(* PLC project LMM.project, Inovance company InoProShop(V1.9.1.6) InoProShop(V1.9.1.6) *)
(* stored: creationDateTime 2026-07-16T22:05:55.4194763, modificationDateTime 2026-07-16T22:05:33.9327845 *)

VAR_GLOBAL  (* GVL *)
  StartBtn AT %IX1.6 : BOOL;  (* 【面板启动】AT %IX1.6 → HMI_xStart/HMI_xEnable（上升沿 STOP→RUN） *)
  StopBtn AT %IX1.4 : BOOL;  (* 【面板停止】AT %IX1.4 → HMI_xStop *)
  ResetBtn : BOOL;  (* 【面板复位】→ HMI_xStopHold3s（错误复位脉冲）；地址现场可另绑 *)
  EStop AT %IX0.4 : BOOL;  (* 【面板急停】AT %IX0.4 正常=TRUE 按下=FALSE → 直通 HMI_xEStop *)
  StopLamp AT %QX0.6 : BOOL;  (* 【停止指示灯】AT %QX0.6 ← Dev_xStop（停止/待机） *)
  StartLamp AT %QX0.7 : BOOL;  (* 【启动/运行指示灯】AT %QX0.7 ← Dev_xRun（正在运行） *)
  JogVel : REAL;  (* 面板点动速度 → 桥接到 HMI_rJogVel* *)
  JogFwd : BOOL;  (* 面板前进 → 按 X 模式映射到 Sync/Diff/独立点动+ *)
  JogBwd : BOOL;  (* 面板后退 → 按 X 模式映射到 Sync/Diff/独立点动- *)
  JogUp : BOOL;  (* 面板上 → HMI_xJogZPos *)
  JogDown : BOOL;  (* 面板下 → HMI_xJogZNeg *)
  JogRight : BOOL;  (* 面板右 → HMI_xJogYPos *)
  JogLeft : BOOL;  (* 面板左 → HMI_xJogYNeg *)
  JogClockAdd : BOOL;  (* 顺时针 *)
  JogClockMis : BOOL;  (* 逆时针 *)
  JogACC : REAL;  (* 点动加速度 → AxisCmd_rAcc *)
  JogDEC : REAL;  (* 点动减速度 → AxisCmd_rDec *)
  HomeReq : BOOL;  (* 面板回零 → HMI_xHomeReqY/Z *)
  CaliForReq : BOOL;  (* 重力标定 *)
  ClearBruch : BOOL;  (* 毛刷清洗 *)
  yLength : REAL;  (* 龙门跨距/Y长度设定 4..6m → HMI_rWheelBase *)
  HMI_xEStop : BOOL;  (* 【急停】TRUE=未按下(正常)；FALSE=急停按下。可按可松，锁存由Logic保持 *)
  HMI_xStop : BOOL;  (* 【设备停止】短按RUN→STOP；长按3s故障复位 *)
  HMI_xStopHold3s : BOOL;  (* 【停止长按满3s脉冲】清急停锁存+轴错误复位+下使能 *)
  HMI_xEnable : BOOL;  (* 【使能/启动别名】与HMI_xStart等效；上升沿STOP→RUN *)
  Dev_xError : BOOL;  (* 【内部故障态】 *)
  Dev_xRun : BOOL;  (* 【内部运行态】 *)
  Dev_xStop : BOOL;  (* 【内部停机态】 *)
  eDevState : INT;  (* 【设备状态】0STOP 1RUN 2ERROR *)
  HMI_xDevError : BOOL;  (* 【故障灯设备级】 *)
  HMI_xDevRun : BOOL;  (* 【运行灯】 *)
  HMI_xDevStop : BOOL;  (* 【停机灯】 *)
  HMI_eOpMode : INT;  (* 【运行方式】0手动 1自动；配合Run灯 *)
  HMI_eDevState : INT;  (* 【设备状态码】0=STOP 1=RUN 2=ERROR *)
  HMI_xStart : BOOL;  (* 【设备启动】瞬时；上升沿STOP→RUN *)
  HMI_xJogYPos : BOOL;  (* 【Y点动+】TRUE移动 FALSE暂停；受限位/Z忙 *)
  HMI_xJogYNeg : BOOL;  (* 【Y点动-】TRUE移动 FALSE暂停 *)
  HMI_xJogZPos : BOOL;  (* 【Z点动+】TRUE移动 FALSE暂停 *)
  HMI_xJogZNeg : BOOL;  (* 【Z点动-】TRUE移动 FALSE暂停 *)
  HMI_xJogRPos : BOOL;  (* 【R点动+】预留；M5未就绪无效 *)
  HMI_xJogRNeg : BOOL;  (* 【R点动-】预留 *)
  HMI_rJogVelX : REAL := 0.4;  (* 【X点动速度】龙门X基速设定 *)
  AxisCmd_rSpinVel : REAL := 0.0;
  HMI_rJogVelR : REAL := 0.2;  (* 【R轴手动速度】 *)
  HMI_rSpinVel : REAL := 0.3;  (* 【X轴旋转速度】 *)
  HMI_rJogVelY : REAL := 0.4;  (* 【Y点动速度】 *)
  HMI_rJogVelZ : REAL := 0.4;  (* 【Z点动速度】 *)
  HMI_rWheelBase : REAL := 5.0;  (* 【龙门跨距=Y行程】单位m，合法范围4..6；自动Y走距用此值 *)
  xEStopLatched : BOOL;  (* 【急停锁存】按下急停置位；仅长按停止复位可清 *)
  xEnablePermit : BOOL;  (* 【使能许可】急停未触发且无锁存且无故障；≠已上使能 *)
  xFaultAggregate : BOOL;  (* 【故障汇总】任轴Fault *)
  xIlk_BlockYPlus : BOOL;  (* 【联锁禁Y+】由Y+限位派生 *)
  xIlk_BlockYNeg : BOOL;  (* 【联锁禁Y-】由Y-限位派生 *)
  xIlk_BlockZPlus : BOOL;  (* 【联锁禁Z+】由Z+限位派生 *)
  xIlk_BlockZNeg : BOOL;  (* 【联锁禁Z-】由Z-限位派生 *)
  xIlk_BlockYWhenZ : BOOL;  (* 【Z动禁Y】Z运动中禁止Y点动 *)
  xM5Ready : BOOL;  (* 【第5轴就绪】FALSE=忽略R轴 *)
  HMI_xLampEStop : BOOL;  (* 【急停灯】HMI读；锁存或按钮仍按下 *)
  HMI_xLampEnableOk : BOOL;  (* 【使能/运行灯】=设备RUN *)
  HMI_xLampFault : BOOL;  (* 【轴故障灯】 *)
  eOpMode : INT;  (* 【运行模式】0=手动Manual（本期固定） *)
  iAlarmID : INT;  (* 【内部报警号】Logic判定后拷贝到HMI_iAlarmShow *)
  HMI_iAlarmShow : INT;  (* 【报警号】0无；1001急停；1002故障；1003限位；1004无许可；1099R未就绪 *)
  I_xLimYPos : BOOL;  (* 【Y正限位】物理输入，地址%I* TBD *)
  I_xLimYNeg : BOOL;  (* 【Y负限位】物理输入 *)
  I_xHomeY : BOOL;  (* 【Y原点】物理输入 *)
  I_xLimZPos : BOOL;  (* 【Z正限位】物理输入 *)
  I_xLimZNeg : BOOL;  (* 【Z负限位】物理输入 *)
  I_xHomeZ : BOOL;  (* 【Z原点】物理输入 *)
  I_xLimRPos : BOOL;  (* 【R正限位】预留 *)
  I_xLimRNeg : BOOL;  (* 【R负限位】预留 *)
  I_xHomeR : BOOL;  (* 【R原点】预留 *)
  AxisCmd_xPower : BOOL;  (* 【轴使能命令】仅设备RUN时TRUE *)
  AxisCmd_xJogYPos : BOOL;  (* 【Y点动+命令】含限位/Z忙门控 *)
  AxisCmd_xJogYNeg : BOOL;  (* 【Y点动-命令】 *)
  AxisCmd_xJogZPos : BOOL;  (* 【Z点动+命令】 *)
  AxisCmd_xJogZNeg : BOOL;  (* 【Z点动-命令】 *)
  AxisCmd_xJogRPos : BOOL;  (* 【R点动+命令】预留 *)
  AxisCmd_xJogRNeg : BOOL;  (* 【R点动-命令】预留 *)
  AxisCmd_xStopAll : BOOL;  (* 【全停】急停/停止/故障时TRUE *)
  AxisCmd_xResetFault : BOOL;  (* 【错误复位脉冲】一拍TRUE→各轴MC_Reset *)
  AxisCmd_rWheelBase : REAL;  (* 【跨距L命令】限幅4..6m *)
  AxisCmd_rJogVelX : REAL;  (* 【X点动速度命令】 *)
  AxisCmd_rJogVelY : REAL;  (* 【Y点动速度命令】 *)
  AxisCmd_rJogVelZ : REAL;  (* 【Z点动速度命令】 *)
  AxisCmd_rJogVelR : REAL;  (* 【R点动速度命令】预留 *)
  AxisCmd_rAcc : REAL;  (* 【加速度】 *)
  AxisCmd_rDec : REAL;  (* 【减速度】 *)
  AxisFb_rVelCmdM1 : REAL;  (* 【M1速度指令反馈】供HMI显示 *)
  AxisFb_rVelCmdM2 : REAL;  (* 【M2速度指令反馈】 *)
  AxisFb_rPosM1 : REAL;  (* 【M1实际位置】 *)
  AxisFb_rPosM2 : REAL;  (* 【M2实际位置】 *)
  AxisFb_rPosY : REAL;  (* 【Y实际位置】 *)
  AxisFb_rPosZ : REAL;  (* 【Z实际位置】 *)
  AxisFb_rPosR : REAL;  (* 【R实际位置】预留 *)
  AxisFb_xStandstill1 : BOOL;  (* 【M1静止】 *)
  AxisFb_xStandstill2 : BOOL;  (* 【M2静止】 *)
  AxisFb_xStandstillY : BOOL;  (* 【Y静止】 *)
  AxisFb_xStandstillZ : BOOL;  (* 【Z静止】 *)
  AxisFb_xStandstillR : BOOL;  (* 【R静止】预留 *)
  AxisFb_xMovingM1 : BOOL;  (* 【M1运动中】 *)
  AxisFb_xMovingM2 : BOOL;  (* 【M2运动中】 *)
  AxisFb_xMovingY : BOOL;  (* 【Y运动中】 *)
  AxisFb_xMovingZ : BOOL;  (* 【Z运动中】 *)
  AxisFb_xMovingR : BOOL;  (* 【R运动中】预留 *)
  AxisFb_xPoweredM1 : BOOL;  (* 【M1已使能】驱动功率级就绪，HMI灯 *)
  AxisFb_xPoweredM2 : BOOL;  (* 【M2已使能】 *)
  AxisFb_xPoweredY : BOOL;  (* 【Y已使能】 *)
  AxisFb_xPoweredZ : BOOL;  (* 【Z已使能】 *)
  AxisFb_xPoweredR : BOOL;  (* 【R已使能】预留 *)
  AxisFb_xHomedY : BOOL;  (* 【Y已回零】 *)
  AxisFb_xHomedZ : BOOL;  (* 【Z已回零】 *)
  AxisFb_xHomedR : BOOL;  (* 【R已回零】预留 *)
  AxisFb_xFaultM1 : BOOL;  (* 【M1故障】 *)
  AxisFb_xFaultM2 : BOOL;  (* 【M2故障】 *)
  AxisFb_xFaultY : BOOL;  (* 【Y故障】 *)
  AxisFb_xFaultZ : BOOL;  (* 【Z故障】 *)
  AxisFb_xFaultR : BOOL;  (* 【R故障】预留 *)
  AxisFb_xReady : BOOL;  (* 【轴就绪】四轴无故障、可参与运动 *)
  HMI_xAutoMode : BOOL;  (* 【自动模式】TRUE自动 FALSE手动 *)
  HMI_xJogXPos : BOOL;  (* 【X+】同步直行 *)
  HMI_xJogXNeg : BOOL;  (* 【X-】 *)
  HMI_xSpinLeft : BOOL;  (* 【左旋转】 *)
  HMI_xSpinRight : BOOL;  (* 【右旋转】 *)
  HMI_xAutoStart : BOOL;  (* 【自动启动】 *)
  HMI_xAutoAbort : BOOL;  (* 【自动中止】 *)
  HMI_rAutoDistX : REAL;  (* 【自动X距离】 *)
  HMI_rAutoVelX : REAL;  (* 【自动X速度】 *)
  HMI_rAutoVelY : REAL;  (* 【自动Y速度】 *)
  HMI_rAutoVelZ : REAL;  (* 【自动Z速度】 *)
  HMI_rForceSet : REAL;  (* 【力设定N】 *)
  HMI_xForceSimEnable : BOOL;  (* 【力模拟使能】 *)
  HMI_rForceSim : REAL;  (* 【力模拟值N】 *)
  HMI_iAutoStepShow : INT;  (* 【自动步号】 *)
  HMI_xAutoBusy : BOOL;  (* 【自动忙】 *)
  HMI_xAutoDone : BOOL;  (* 【自动完成】 *)
  HMI_rForceShow : REAL;  (* 【力实际N】 *)
  Tcp_xConnected : BOOL;  (* 【TCP】已连接 *)
  Tcp_xTimeout : BOOL;  (* 【TCP】通讯超时 *)
  Tcp_xOnline : BOOL;  (* 【TCP】Connected且未超时 *)
  Tcp_xEStop : BOOL := TRUE;  (* 【TCP急停影子】默认TRUE；与面板AND合成 *)
  Tcp_xStop : BOOL;
  Tcp_xStopHold3s : BOOL;
  Tcp_xStart : BOOL;
  Tcp_xEnable : BOOL;
  Tcp_xAutoMode : BOOL;
  Tcp_xJogXPos : BOOL;
  Tcp_xJogXNeg : BOOL;
  Tcp_xSpinLeft : BOOL;
  Tcp_xSpinRight : BOOL;
  Tcp_xJogYPos : BOOL;
  Tcp_xJogYNeg : BOOL;
  Tcp_xJogZPos : BOOL;
  Tcp_xJogZNeg : BOOL;
  Tcp_xJogRPos : BOOL;
  Tcp_xJogRNeg : BOOL;
  Tcp_rJogVelX : REAL := 0.4;
  Tcp_rSpinVel : REAL := 0.3;
  Tcp_rJogVelY : REAL := 0.3;
  Tcp_rJogVelZ : REAL := 0.2;
  Tcp_rJogVelR : REAL := 0.2;
  Tcp_xAutoStart : BOOL;
  Tcp_xAutoAbort : BOOL;
  Tcp_rAutoDistX : REAL := 1.0;
  Tcp_rAutoVelX : REAL := 0.4;
  Tcp_rAutoVelY : REAL := 0.3;
  Tcp_rAutoVelZ : REAL := 0.15;
  Tcp_rWheelBase : REAL := 5.0;
  Tcp_rForceSet : REAL := 100.0;
  Tcp_xForceSimEnable : BOOL := TRUE;
  Tcp_rForceSim : REAL;
  Tcp_uiPort : UINT := 9100;  (* 【TCP监听端口】默认9100 *)
  iAutoStep : INT;  (* 【自动步】0Idle..5Done *)
  rForceAct : REAL;  (* 【实际力N】 *)
  rForceKp : REAL;  (* 【恒力Kp】 *)
  AxisCmd_xJogXPos : BOOL;  (* 【Axis X+】 *)
  AxisCmd_xJogXNeg : BOOL;  (* 【Axis X-】 *)
  AxisCmd_xSpinLeft : BOOL;  (* 【Axis 左旋】 *)
  AxisCmd_xSpinRight : BOOL;  (* 【Axis 右旋】 *)
  AxisCmd_xMoveRelX : BOOL;  (* 【Axis X相对】 *)
  AxisCmd_rMoveDistX : REAL;  (* 【X相对距离】 *)
  AxisCmd_rMoveVelX : REAL;  (* 【X相对速度】 *)
  AxisCmd_xMoveRelY : BOOL;  (* 【Axis Y相对】 *)
  AxisCmd_rMoveDistY : REAL;  (* 【Y相对距离】 *)
  AxisCmd_rMoveVelY : REAL;  (* 【Y相对速度】 *)
  AxisCmd_rZVelCmd : REAL;  (* 【Z速度指令】 *)
  AxisCmd_xUseZVelCmd : BOOL;  (* 【使用Z速度指令】 *)
  AxisCmd_xHoldR : BOOL;  (* 【R保持】 *)
  AxisCmd_rRHoldPos : REAL;  (* 【R保持角】 *)
  AxisFb_xMoveDoneX : BOOL;  (* 【X相对到位】 *)
  AxisFb_xMoveDoneY : BOOL;  (* 【Y相对到位】 *)
END_VAR

PROGRAM PRG_Axis_Control
  VAR
    fbM1 : FB_Servo;
    fbM2 : FB_Servo;
    fbY : FB_Servo;
    fbZ : FB_Servo;
    fbXDiff : FB_XDiff;
    xPair : BOOL;
    eModeX : INT;
    xDiffPos : BOOL;
    xDiffNeg : BOOL;
    rXVel : REAL;
  END_VAR

            (*==============================================================================
 * PRG_Axis_Control — 运动独立任务（AxisTask）
 * 仅通过 GVL_AxisCmd 输入 / GVL_AxisFb 输出；禁止被外部 CALL
 * 轴绑定：Axis=M1, Axis_1=M2, Axis_2=Y, Axis_3=Z
 *============================================================================*)

(* X：同步直行 / 左右旋；VelX 与 SpinVel 分开 *)
eModeX := 0;
xDiffPos := FALSE; xDiffNeg := FALSE;
IF AxisCmd_xSpinLeft XOR AxisCmd_xSpinRight THEN
	eModeX := 2;
	xDiffPos := AxisCmd_xSpinLeft;
	xDiffNeg := AxisCmd_xSpinRight;
	rXVel := AxisCmd_rSpinVel;
ELSIF AxisCmd_xJogXPos XOR AxisCmd_xJogXNeg THEN
	eModeX := 1;
	rXVel := AxisCmd_rJogVelX;
ELSE
	rXVel := 0.0;
END_IF;

fbXDiff(
	eMode := eModeX,
	eDiffFunc := 1,
	xJogSyncPos := AxisCmd_xJogXPos,
	xJogSyncNeg := AxisCmd_xJogXNeg,
	xJogDiffPos := xDiffPos,
	xJogDiffNeg := xDiffNeg,
	xStop := AxisCmd_xStopAll,
	xEnable := AxisCmd_xPower,
	rJogVel := rXVel,
	rDiffDelta := 0.0,
	rTurnOmega := 0.0,
	rWheelBase := AxisCmd_rWheelBase
);
xPair := fbXDiff.xUsePairVel;

IF xPair THEN
	(* 成对模式：用 FB_XDiff 输出的有符号速度 *)
	fbM1(
		Axis := _MC_Axis[1],
		xEnable := AxisCmd_xPower,
		xJogPos := FALSE, xJogNeg := FALSE,
		xStop := AxisCmd_xStopAll,
		xResetFault := AxisCmd_xResetFault,
		xHome := FALSE,
		xUseVelCmd := TRUE,
		rVelCmd := fbXDiff.rVelCmdM1,
		rJogVel := rXVel,
		rAcc := AxisCmd_rAcc,
		rDec := AxisCmd_rDec
	);
	fbM2(
		Axis := _MC_Axis[2],
		xEnable := AxisCmd_xPower,
		xJogPos := FALSE, xJogNeg := FALSE,
		xStop := AxisCmd_xStopAll,
		xResetFault := AxisCmd_xResetFault,
		xHome := FALSE,
		xUseVelCmd := TRUE,
		rVelCmd := fbXDiff.rVelCmdM2,
		rJogVel := rXVel,
		rAcc := AxisCmd_rAcc,
		rDec := AxisCmd_rDec
	);
	AxisFb_rVelCmdM1 := fbXDiff.rVelCmdM1;
	AxisFb_rVelCmdM2 := fbXDiff.rVelCmdM2;
ELSE
	(* 无 X 命令：两侧保持上电待机 *)
	fbM1(
		Axis := _MC_Axis[1],
		xEnable := AxisCmd_xPower,
		xJogPos := FALSE, xJogNeg := FALSE,
		xStop := AxisCmd_xStopAll,
		xResetFault := AxisCmd_xResetFault,
		xHome := FALSE,
		xUseVelCmd := FALSE,
		rVelCmd := 0.0,
		rJogVel := AxisCmd_rJogVelX,
		rAcc := AxisCmd_rAcc,
		rDec := AxisCmd_rDec
	);
	fbM2(
		Axis := _MC_Axis[2],
		xEnable := AxisCmd_xPower,
		xJogPos := FALSE, xJogNeg := FALSE,
		xStop := AxisCmd_xStopAll,
		xResetFault := AxisCmd_xResetFault,
		xHome := FALSE,
		xUseVelCmd := FALSE,
		rVelCmd := 0.0,
		rJogVel := AxisCmd_rJogVelX,
		rAcc := AxisCmd_rAcc,
		rDec := AxisCmd_rDec
	);
	AxisFb_rVelCmdM1 := 0.0;
	AxisFb_rVelCmdM2 := 0.0;
END_IF;

(* Y / Z *)
fbY(
	Axis := _MC_Axis[3],
	xEnable := AxisCmd_xPower,
	xJogPos := AxisCmd_xJogYPos,
	xJogNeg := AxisCmd_xJogYNeg,
	xStop := AxisCmd_xStopAll,
	xResetFault := AxisCmd_xResetFault,
	xHome := FALSE,
	xUseVelCmd := FALSE,
	rVelCmd := 0.0,
	rJogVel := AxisCmd_rJogVelY,
	rAcc := AxisCmd_rAcc,
	rDec := AxisCmd_rDec
);
fbZ(
	Axis := _MC_Axis[4],
	xEnable := AxisCmd_xPower,
	xJogPos := AxisCmd_xJogZPos,
	xJogNeg := AxisCmd_xJogZNeg,
	xStop := AxisCmd_xStopAll,
	xResetFault := AxisCmd_xResetFault,
	xHome := FALSE,
	xUseVelCmd := FALSE,
	rVelCmd := 0.0,
	rJogVel := AxisCmd_rJogVelZ,
	rAcc := AxisCmd_rAcc,
	rDec := AxisCmd_rDec
);

(* ---------- 写反馈区（仅本任务可写） ---------- *)
AxisFb_rPosM1 := fbM1.rActPos;
AxisFb_rPosM2 := fbM2.rActPos;
AxisFb_rPosY := fbY.rActPos;
AxisFb_rPosZ := fbZ.rActPos;
AxisFb_xMovingM1 := fbM1.xMoving;
AxisFb_xMovingM2 := fbM2.xMoving;
AxisFb_xMovingY := fbY.xMoving;
AxisFb_xMovingZ := fbZ.xMoving;
AxisFb_xPoweredM1 := fbM1.xPowered;
AxisFb_xPoweredM2 := fbM2.xPowered;
AxisFb_xPoweredY := fbY.xPowered;
AxisFb_xPoweredZ := fbZ.xPowered;
AxisFb_xFaultM1 := fbM1.xFault;
AxisFb_xFaultM2 := fbM2.xFault;
AxisFb_xFaultY := fbY.xFault;
AxisFb_xFaultZ := fbZ.xFault;
AxisFb_xHomedY := fbY.xHomed;
AxisFb_xHomedZ := fbZ.xHomed;
AxisFb_xStandstill1 := fbM1.xStandstill;
AxisFb_xStandstill2 := fbM2.xStandstill;
AxisFb_xStandstillY := fbY.xStandstill;
AxisFb_xStandstillZ := fbZ.xStandstill;
AxisFb_xReady := NOT (fbM1.xFault OR fbM2.xFault OR fbY.xFault OR fbZ.xFault);

          
END_PROGRAM

FUNCTION_BLOCK FB_XDiff
  VAR_INPUT
    eMode : INT;
    eDiffFunc : INT;
    xJogSyncPos : BOOL;
    xJogSyncNeg : BOOL;
    xJogDiffPos : BOOL;
    xJogDiffNeg : BOOL;
    xStop : BOOL;
    xEnable : BOOL;
    rJogVel : REAL;
    rDiffDelta : REAL;
    rTurnOmega : REAL;
    rWheelBase : REAL;
  END_VAR
  VAR_OUTPUT
    rVelCmdM1 : REAL;
    rVelCmdM2 : REAL;
    xActive : BOOL;
    xUsePairVel : BOOL;
    xWheelBaseOk : BOOL;
  END_VAR

            (*==============================================================================
 * FB_XDiff — 龙门 X 双驱速度合成（仅 Axis 任务内使用）
 * eMode: 0=独立  1=同步同速平移  2=差速（子功能见 eDiffFunc）
 * eDiffFunc: 0=纠偏  1=原地旋转(一正一反)  2=差速拐弯
 * 跨距 rWheelBase: 4..6 m；X 运动方向与 Y 垂直
 *============================================================================*)

(* 输出清零 *)
rVelCmdM1 := 0.0;
rVelCmdM2 := 0.0;
xUsePairVel := FALSE;
xActive := FALSE;
(* 跨距合法性 *)
xWheelBaseOk := (rWheelBase >= 4.0) AND (rWheelBase <= 6.0);

(* 未使能 / 停止 / 独立模式：不合成成对速度 *)
IF NOT xEnable OR xStop OR eMode = 0 THEN
	RETURN;
END_IF;

(* ---------- Sync：两侧同速，龙门沿 X 平移 ---------- *)
IF eMode = 1 THEN
	IF xJogSyncPos XOR xJogSyncNeg THEN
		xUsePairVel := TRUE;
		xActive := TRUE;
		IF xJogSyncPos THEN
			rVelCmdM1 := rJogVel;
		ELSE
			rVelCmdM1 := -rJogVel;
		END_IF;
		rVelCmdM2 := rVelCmdM1; (* 同速 *)
	END_IF;
	RETURN;
END_IF;

(* ---------- Diff：需有方向键 ---------- *)
IF NOT (xJogDiffPos XOR xJogDiffNeg) THEN
	RETURN;
END_IF;

(* 原地旋转 / 差速拐弯依赖合法跨距 *)
IF (eDiffFunc = 1 OR eDiffFunc = 2) AND NOT xWheelBaseOk THEN
	RETURN;
END_IF;

xUsePairVel := TRUE;
xActive := TRUE;

CASE eDiffFunc OF
	0: (* 纠偏：同向 V±Δ，扶正龙门 *)
		IF xJogDiffPos THEN
			rVelCmdM1 := rJogVel + rDiffDelta;
			rVelCmdM2 := rJogVel - rDiffDelta;
		ELSE
			rVelCmdM1 := -(rJogVel + rDiffDelta);
			rVelCmdM2 := -(rJogVel - rDiffDelta);
		END_IF;

	1: (* 原地旋转：M1/M2 一正一反，转角度 *)
		IF ABS(rTurnOmega) > 1.0E-6 THEN
			rVelCmdM1 := rTurnOmega * rWheelBase * 0.5;
		ELSE
			rVelCmdM1 := rJogVel;
		END_IF;
		rVelCmdM2 := -rVelCmdM1;
		IF xJogDiffNeg THEN
			rVelCmdM1 := -rVelCmdM1;
			rVelCmdM2 := -rVelCmdM2;
		END_IF;

	2: (* 差速拐弯：两侧同向为主，速度差，可边走边弯 *)
		IF ABS(rTurnOmega) > 1.0E-6 THEN
			rVelCmdM1 := rJogVel + rTurnOmega * rWheelBase * 0.5;
			rVelCmdM2 := rJogVel - rTurnOmega * rWheelBase * 0.5;
		ELSE
			rVelCmdM1 := rJogVel + rDiffDelta;
			rVelCmdM2 := rJogVel - rDiffDelta;
		END_IF;
		IF xJogDiffNeg THEN
			rVelCmdM1 := -rVelCmdM1;
			rVelCmdM2 := -rVelCmdM2;
		END_IF;

ELSE
	xUsePairVel := FALSE;
	xActive := FALSE;
END_CASE;

          
END_FUNCTION_BLOCK

PROGRAM PLC_PRG

            (*==============================================================================
 * PLC_PRG — 主任务入口（MainTask）
 * 只调用逻辑程序；禁止在此 CALL PRG_Axis_Control（轴控在独立 AxisTask）
 *============================================================================*)
PRG_TcpHmi();
PRG_Logic();

          
END_PROGRAM

PROGRAM PRG_Logic
  VAR
    tonHold : TON;
    tonResetHold : TON;
    xResetPulse : BOOL;
    xResetPrev : BOOL;
    xStartEdge : BOOL;
    xStartPrev : BOOL;
    xStopEdge : BOOL;
    xStopPrev : BOOL;
    xPostResetHold : BOOL;
    xAutoStartPrev : BOOL;
    xAutoStartEdge : BOOL;
    rRHold : REAL;
    xMoveXSent : BOOL;
    xMoveYSent : BOOL;
    xBridgeInited : BOOL;
  END_VAR

            (*==============================================================================
 * PRG_Logic — 设备态 / 手动裁定 / 自动步序 / 恒力
 * 禁止 CALL Axis / FB_Servo / FB_XDiff
 *============================================================================*)

(* —— 面板 ∨ TCP 影子 → HMI（见 docs/plc/TCP_HMI.md）—— *)
Tcp_xOnline := Tcp_xConnected AND NOT Tcp_xTimeout;
HMI_xEStop := EStop AND Tcp_xEStop;
HMI_xStop := StopBtn OR Tcp_xStop;
HMI_xStart := StartBtn OR Tcp_xStart;
HMI_xEnable := StartBtn OR Tcp_xEnable OR Tcp_xStart;
HMI_xStopHold3s := ResetBtn OR Tcp_xStopHold3s;
IF Tcp_xOnline THEN
	HMI_xAutoMode := Tcp_xAutoMode;
	HMI_xForceSimEnable := Tcp_xForceSimEnable;
END_IF;
HMI_xJogXPos := JogFwd OR Tcp_xJogXPos;
HMI_xJogXNeg := JogBwd OR Tcp_xJogXNeg;
HMI_xSpinLeft := Tcp_xSpinLeft;
HMI_xSpinRight := Tcp_xSpinRight;
HMI_xJogYPos := JogRight OR Tcp_xJogYPos;
HMI_xJogYNeg := JogLeft OR Tcp_xJogYNeg;
HMI_xJogZPos := JogUp OR Tcp_xJogZPos;
HMI_xJogZNeg := JogDown OR Tcp_xJogZNeg;
HMI_xJogRPos := Tcp_xJogRPos;
HMI_xJogRNeg := Tcp_xJogRNeg;
HMI_xAutoStart := Tcp_xAutoStart;
HMI_xAutoAbort := Tcp_xAutoAbort;
IF Tcp_xOnline THEN
	HMI_rJogVelX := Tcp_rJogVelX;
	HMI_rSpinVel := Tcp_rSpinVel;
	HMI_rJogVelY := Tcp_rJogVelY;
	HMI_rJogVelZ := Tcp_rJogVelZ;
	HMI_rJogVelR := Tcp_rJogVelR;
	HMI_rAutoDistX := Tcp_rAutoDistX;
	HMI_rAutoVelX := Tcp_rAutoVelX;
	HMI_rAutoVelY := Tcp_rAutoVelY;
	HMI_rAutoVelZ := Tcp_rAutoVelZ;
	HMI_rWheelBase := Tcp_rWheelBase;
	HMI_rForceSet := Tcp_rForceSet;
	HMI_rForceSim := Tcp_rForceSim;
ELSE
	HMI_rJogVelX := JogVel;
	HMI_rJogVelY := JogVel;
	HMI_rJogVelZ := JogVel;
END_IF;

(* —— 急停 / 复位 —— *)
IF NOT HMI_xEStop THEN xEStopLatched := TRUE; END_IF;
tonHold(IN := HMI_xStop AND HMI_xEStop, PT := T#3S);
xResetPulse := (HMI_xStopHold3s OR tonHold.Q) AND NOT xResetPrev;
xResetPrev := HMI_xStopHold3s OR tonHold.Q;
IF xResetPulse THEN
	xEStopLatched := FALSE;
	AxisCmd_xResetFault := TRUE;
	eDevState := 0;
	xPostResetHold := TRUE;
	iAutoStep := 0;
ELSE
	AxisCmd_xResetFault := FALSE;
END_IF;

xFaultAggregate := AxisFb_xFaultM1 OR AxisFb_xFaultM2 OR AxisFb_xFaultY OR AxisFb_xFaultZ
	OR (xM5Ready AND AxisFb_xFaultR);
xEnablePermit := HMI_xEStop AND NOT xEStopLatched AND NOT xFaultAggregate;
IF HMI_xAutoMode THEN eOpMode := 1; ELSE eOpMode := 0; END_IF;
HMI_eOpMode := eOpMode;

tonResetHold(IN := xPostResetHold, PT := T#2S);
IF NOT xFaultAggregate AND HMI_xEStop AND NOT xEStopLatched THEN
	xPostResetHold := FALSE;
ELSIF tonResetHold.Q OR NOT HMI_xEStop OR xEStopLatched THEN
	xPostResetHold := FALSE;
END_IF;

xStartEdge := (HMI_xStart OR HMI_xEnable) AND NOT xStartPrev;
xStartPrev := HMI_xStart OR HMI_xEnable;
xStopEdge := HMI_xStop AND NOT xStopPrev;
xStopPrev := HMI_xStop;

IF xResetPulse THEN
	eDevState := 0;
ELSIF NOT HMI_xEStop OR xEStopLatched THEN
	eDevState := 2;
ELSIF xFaultAggregate AND NOT xPostResetHold THEN
	eDevState := 2;
ELSIF eDevState = 2 THEN
	;
ELSIF xStopEdge AND NOT tonHold.Q THEN
	eDevState := 0;
	iAutoStep := 0;
ELSIF xStartEdge AND eDevState = 0 AND xEnablePermit THEN
	eDevState := 1;
ELSIF xStartEdge AND eDevState = 0 AND NOT xEnablePermit THEN
	iAlarmID := 1004;
END_IF;

Dev_xStop := (eDevState = 0);
Dev_xRun := (eDevState = 1);
Dev_xError := (eDevState = 2);
HMI_eDevState := eDevState;
HMI_xDevStop := Dev_xStop;
HMI_xDevRun := Dev_xRun;
HMI_xDevError := Dev_xError;

IF HMI_xForceSimEnable THEN
	rForceAct := HMI_rForceSim;
END_IF;
HMI_rForceShow := rForceAct;
IF rForceKp < 1.0E-6 THEN rForceKp := 1.0; END_IF;

xIlk_BlockYPlus := I_xLimYPos; xIlk_BlockYNeg := I_xLimYNeg;
xIlk_BlockZPlus := I_xLimZPos; xIlk_BlockZNeg := I_xLimZNeg;
xIlk_BlockYWhenZ := FALSE;

AxisCmd_xStopAll := (eDevState <> 1) OR HMI_xStop OR HMI_xAutoAbort;
AxisCmd_xPower := (eDevState = 1);
AxisCmd_rJogVelX := HMI_rJogVelX;
AxisCmd_rSpinVel := HMI_rSpinVel;
AxisCmd_rJogVelY := HMI_rJogVelY;
AxisCmd_rJogVelZ := HMI_rJogVelZ;
AxisCmd_rJogVelR := HMI_rJogVelR;
AxisCmd_rWheelBase := LIMIT(4.0, HMI_rWheelBase, 6.0);
AxisCmd_rAcc := JogACC;
AxisCmd_rDec := JogDEC;
IF AxisCmd_rAcc < 1.0 THEN AxisCmd_rAcc := 100.0; END_IF;
IF AxisCmd_rDec < 1.0 THEN AxisCmd_rDec := 100.0; END_IF;

AxisCmd_xJogXPos := FALSE; AxisCmd_xJogXNeg := FALSE;
AxisCmd_xSpinLeft := FALSE; AxisCmd_xSpinRight := FALSE;
AxisCmd_xJogYPos := FALSE; AxisCmd_xJogYNeg := FALSE;
AxisCmd_xJogZPos := FALSE; AxisCmd_xJogZNeg := FALSE;
AxisCmd_xJogRPos := FALSE; AxisCmd_xJogRNeg := FALSE;
AxisCmd_xUseZVelCmd := FALSE; AxisCmd_rZVelCmd := 0.0;
AxisCmd_xMoveRelX := FALSE; AxisCmd_xMoveRelY := FALSE;
AxisCmd_xHoldR := FALSE;

xAutoStartEdge := HMI_xAutoStart AND NOT xAutoStartPrev;
xAutoStartPrev := HMI_xAutoStart;

IF Dev_xError OR HMI_xAutoAbort OR (eDevState <> 1) THEN
	iAutoStep := 0;
	HMI_xAutoBusy := FALSE;
END_IF;

(* ===== 手动：仅 RUN + 手动模式 ===== *)
IF Dev_xRun AND (eOpMode = 0) AND NOT HMI_xStop THEN
	IF HMI_xSpinLeft XOR HMI_xSpinRight THEN
		AxisCmd_xSpinLeft := HMI_xSpinLeft;
		AxisCmd_xSpinRight := HMI_xSpinRight;
	ELSIF HMI_xJogXPos XOR HMI_xJogXNeg THEN
		AxisCmd_xJogXPos := HMI_xJogXPos;
		AxisCmd_xJogXNeg := HMI_xJogXNeg;
	END_IF;
	AxisCmd_xJogYPos := HMI_xJogYPos AND NOT xIlk_BlockYPlus;
	AxisCmd_xJogYNeg := HMI_xJogYNeg AND NOT xIlk_BlockYNeg;
	AxisCmd_xJogZPos := HMI_xJogZPos AND NOT xIlk_BlockZPlus;
	AxisCmd_xJogZNeg := HMI_xJogZNeg AND NOT xIlk_BlockZNeg;
	IF xM5Ready THEN
		AxisCmd_xJogRPos := HMI_xJogRPos;
		AxisCmd_xJogRNeg := HMI_xJogRNeg;
	END_IF;
END_IF;

(* ===== 自动 ===== *)
IF Dev_xRun AND (eOpMode = 1) AND NOT HMI_xStop THEN
	IF iAutoStep = 0 AND xAutoStartEdge THEN
		iAutoStep := 1;
		rRHold := AxisFb_rPosR;
		xMoveXSent := FALSE; xMoveYSent := FALSE;
		HMI_xAutoDone := FALSE;
		HMI_xAutoBusy := TRUE;
	END_IF;

	CASE iAutoStep OF
		1: (* MoveX *)
			AxisCmd_xHoldR := TRUE;
			AxisCmd_rRHoldPos := rRHold;
			AxisCmd_rMoveDistX := HMI_rAutoDistX;
			AxisCmd_rMoveVelX := HMI_rAutoVelX;
			AxisCmd_xMoveRelX := TRUE;
			IF AxisFb_xMoveDoneX THEN
				AxisCmd_xMoveRelX := FALSE;
				iAutoStep := 2;
			END_IF;
		2: (* PressZ *)
			AxisCmd_xHoldR := TRUE;
			AxisCmd_rRHoldPos := rRHold;
			AxisCmd_xUseZVelCmd := TRUE;
			IF rForceAct >= HMI_rForceSet THEN
				AxisCmd_rZVelCmd := 0.0;
				iAutoStep := 3;
				xMoveYSent := FALSE;
			ELSE
				AxisCmd_rZVelCmd := -ABS(HMI_rAutoVelZ);
			END_IF;
		3: (* MoveY + 恒力 *)
			AxisCmd_xHoldR := TRUE;
			AxisCmd_rRHoldPos := rRHold;
			AxisCmd_rMoveDistY := AxisCmd_rWheelBase;
			AxisCmd_rMoveVelY := HMI_rAutoVelY;
			AxisCmd_xMoveRelY := TRUE;
			AxisCmd_xUseZVelCmd := TRUE;
			AxisCmd_rZVelCmd := LIMIT(-ABS(HMI_rAutoVelZ),
				rForceKp * (HMI_rForceSet - rForceAct), ABS(HMI_rAutoVelZ));
			IF AxisFb_xMoveDoneY THEN
				AxisCmd_xMoveRelY := FALSE;
				AxisCmd_rZVelCmd := 0.0;
				iAutoStep := 4;
			END_IF;
		4: (* RWobble 占位 *)
			iAutoStep := 5;
		5: (* Done *)
			HMI_xAutoBusy := FALSE;
			HMI_xAutoDone := TRUE;
			iAutoStep := 0;
	END_CASE;
END_IF;

IF Dev_xError THEN
	IF xEStopLatched OR NOT HMI_xEStop THEN
		iAlarmID := 1001;
	ELSE
		iAlarmID := 1002;
	END_IF;
ELSIF iAlarmID <> 1004 THEN
	iAlarmID := 0;
END_IF;

HMI_iAutoStepShow := iAutoStep;
HMI_xLampEStop := xEStopLatched OR NOT HMI_xEStop;
HMI_xLampEnableOk := Dev_xRun;
HMI_xLampFault := xFaultAggregate;
HMI_iAlarmShow := iAlarmID;

StopLamp := Dev_xStop;
StartLamp := Dev_xRun;

          
END_PROGRAM

FUNCTION_BLOCK FB_Servo
  VAR_INPUT
    xEnable : BOOL;
    xJogPos : BOOL;
    xJogNeg : BOOL;
    xStop : BOOL;
    xResetFault : BOOL;
    xHome : BOOL;
    xUseVelCmd : BOOL;
    rVelCmd : REAL;
    rJogVel : REAL;
    rAcc : REAL;
    rDec : REAL;
  END_VAR
  VAR_OUTPUT
    xPowered : BOOL;
    xMoving : BOOL;
    xStandstill : BOOL;
    xHomed : BOOL;
    xFault : BOOL;
    rActPos : LREAL;
  END_VAR
  VAR_IN_OUT
    Axis : AXIS_REF_SM3;
  END_VAR
  VAR
    fbPower : MC_Power;
    fbJog : MC_MoveVelocity;
    fbStop : MC_Stop;
    fbHome : MC_Home;
    fbReset : MC_Reset;
    fbReadStatus : MC_ReadStatus;
    fbReadPos : MC_ReadActualPosition;
    xEnInternal : BOOL;
  END_VAR

            (* 读轴状态 / 实际位置 *)
fbReadStatus(Axis := Axis, Enable := TRUE);
fbReadPos(Axis := Axis, Enable := TRUE);

rActPos := fbReadPos.Position;
xStandstill := fbReadStatus.StandStill;
xMoving := fbReadStatus.DiscreteMotion OR fbReadStatus.ContinuousMotion;

(* 故障汇总：Errorstop + 各 FB.Error（不用 Axis.bError / Operational） *)
xFault := fbReadStatus.Errorstop
	OR fbReadStatus.Error
	OR fbPower.Error
	OR fbJog.Error
	OR fbStop.Error
	OR fbReset.Error;

(* 错误复位脉冲（来自停止钮长按 3s → AxisCmd_xResetFault） *)
fbReset(Axis := Axis, Execute := xResetFault);

(* 内部使能：请求使能且未停且非 Errorstop *)
xEnInternal := xEnable AND NOT xStop AND NOT fbReadStatus.Errorstop;

(* 功率级：Enable 恒 TRUE 以刷新；实际开/关看 bRegulatorOn/bDriveStart *)
fbPower(
	Axis := Axis,
	Enable := TRUE,
	bRegulatorOn := xEnInternal,
	bDriveStart := xEnInternal
);
(* Status=TRUE 表示轴可运动 *)
xPowered := fbPower.Status;

(* ---------- 运动仲裁 ---------- *)
IF xStop OR NOT xEnable OR fbReadStatus.Errorstop THEN
	(* 停止 / 禁使能 / 故障：停速度指令并减速停 *)
	fbJog(Axis := Axis, Execute := FALSE);
	fbHome(Axis := Axis, Execute := FALSE);
	fbStop(Axis := Axis, Execute := TRUE, Deceleration := rDec);

ELSIF xHome THEN
	(* 回零 *)
	fbStop(Axis := Axis, Execute := FALSE);
	fbJog(Axis := Axis, Execute := FALSE);
	fbHome(Axis := Axis, Execute := TRUE);

ELSIF xUseVelCmd THEN
	(* 成对速度模式：使用有符号 rVelCmd（来自 FB_XDiff） *)
	fbStop(Axis := Axis, Execute := FALSE);
	fbHome(Axis := Axis, Execute := FALSE);
	IF ABS(rVelCmd) > 1.0E-6 AND xPowered THEN
		fbJog(Axis := Axis, Execute := TRUE, Velocity := rVelCmd, Acceleration := rAcc, Deceleration := rDec);
	ELSE
		fbJog(Axis := Axis, Execute := FALSE);
	END_IF;

ELSIF xJogPos XOR xJogNeg THEN
	(* 独立 JOG *)
	fbStop(Axis := Axis, Execute := FALSE);
	fbHome(Axis := Axis, Execute := FALSE);
	IF xPowered THEN
		IF xJogPos THEN
			fbJog(Axis := Axis, Execute := TRUE, Velocity := ABS(rJogVel), Acceleration := rAcc, Deceleration := rDec);
		ELSE
			fbJog(Axis := Axis, Execute := TRUE, Velocity := -ABS(rJogVel), Acceleration := rAcc, Deceleration := rDec);
		END_IF;
	ELSE
		fbJog(Axis := Axis, Execute := FALSE);
	END_IF;

ELSE
	(* 空闲 *)
	fbJog(Axis := Axis, Execute := FALSE);
	fbHome(Axis := Axis, Execute := FALSE);
	fbStop(Axis := Axis, Execute := FALSE);
END_IF;

IF fbHome.Done THEN
	xHomed := TRUE;
END_IF;

          
END_FUNCTION_BLOCK

FUNCTION_BLOCK FB_TCPServer
  VAR_INPUT
    i_xEnable : BOOL;
    i_uiPort : UINT;
    i_xSendTrig : BOOL;
    i_strSend : STRING(512);
  END_VAR
  VAR_OUTPUT
    o_xConnected : BOOL;
    o_xRecvNew : BOOL;
    o_strRecv : STRING(512);
    o_uiRecvLen : UINT;
    o_xSendDone : BOOL;
    o_xError : BOOL;
    o_wErrorID : WORD;
  END_VAR
  VAR
    SktTCPServer : SktTCPServer;
    SktTCPSend : SktTCPSend_C;
    SktTCPRecv : SktTCPRecv_C;
    stLocalAddress : ADDRESS;
    stConnectParam : CONNCET_PARAM;
    stConnectInfo : CONNECT_INFO;
    abyRecv : ARRAY[0..511] OF BYTE;
    abySend : ARRAY[0..511] OF BYTE;
    pRecv : POINTER TO BYTE;
    pSend : POINTER TO BYTE;
    xSendPrev : BOOL;
    xRecvReady : BOOL;
    i : INT;
    n : INT;
    uiLen : UINT;
    sOne : STRING(1);
  END_VAR

            (*==============================================================================
 * FB_TCPServer — 汇川 cmphctcpip / SktTCP*
 *
 * 编译错误根因与对策：
 *  C0032 STRING→ADDRESS     : strLocalAddress 用 ADDRESS 结构，勿传 STRING
 *  C0032 CONNECT_INFO→CONNCET_PARAM : Recv/Send 的 stConnect 用 CONNCET_PARAM
 *  C0078 ARRAY OF BYTE      : abyData 传 POINTER（ADR），勿直接传数组
 *
 * 若 ADDRESS 成员名不同：在 InoProShop 对 ADDRESS 按 F2，改下面两行赋值。
 * 常见：strIpAddress/uiPort 或 sIP/wPort 或 strIP/iPort
 *============================================================================*)
o_xRecvNew := FALSE;
o_xSendDone := FALSE;
IF NOT i_xEnable THEN
	o_xConnected := FALSE;
	RETURN;
END_IF;

stLocalAddress.strIpAddress := '0.0.0.0';
stLocalAddress.uiPort := i_uiPort;

SktTCPServer(
	xExecute := i_xEnable,
	diConnectID := DINT#1,
	strLocalAddress := stLocalAddress,
	xDone => ,
	xBusy => ,
	xError => o_xError,
	wErrorID => o_wErrorID,
	stConnectInfo => stConnectInfo);

(* Recv/Send 要 CONNCET_PARAM；与 Server 共用 ConnectID=1 *)
stConnectParam.diConnectID := DINT#1;

o_xConnected := SktTCPServer.xBusy OR SktTCPServer.xDone;

pRecv := ADR(abyRecv);
pSend := ADR(abySend);

SktTCPRecv(
	xEnable := i_xEnable AND o_xConnected,
	xEnCont := TRUE,
	stConnect := stConnectParam,
	abyData := pRecv,
	uiDataSize := UINT#512,
	xDone => ,
	xBusy => ,
	xError => ,
	wErrorID => ,
	xReady => xRecvReady,
	uiCount => o_uiRecvLen,
	eStatus => ,
	stConnectInfo => stConnectInfo);

IF xRecvReady AND (o_uiRecvLen > 0) THEN
	o_xRecvNew := TRUE;
	IF o_uiRecvLen > 512 THEN
		n := 512;
	ELSE
		n := UINT_TO_INT(o_uiRecvLen);
	END_IF;
	o_strRecv := '';
	FOR i := 0 TO (n - 1) DO
		IF (abyRecv[i] = 16#0A) OR (abyRecv[i] = 16#0D) THEN
			EXIT;
		END_IF;
		sOne := CHR(BYTE_TO_DWORD(abyRecv[i]));
		o_strRecv := CONCAT(o_strRecv, sOne);
	END_FOR;
END_IF;

IF i_xSendTrig AND NOT xSendPrev AND (LEN(i_strSend) > 0) THEN
	n := LEN(i_strSend);
	IF n > 512 THEN n := 512; END_IF;
	FOR i := 1 TO n DO
		(* Codesys 字符串下标为 BYTE 码；若编译不过改用 CODE()/ASC() *)
		abySend[i - 1] := i_strSend[i];
	END_FOR;
	uiLen := INT_TO_UINT(n);
	SktTCPSend(
		xExecute := TRUE,
		xEnCont := FALSE,
		stConnect := stConnectParam,
		abyData := pSend,
		uiDataSize := uiLen,
		uiTimeOut := UINT#100,
		xDone => o_xSendDone,
		xBusy => ,
		xError => ,
		wErrorID => ,
		eStatus => ,
		stConnectInfo => );
ELSE
	SktTCPSend(
		xExecute := FALSE,
		xEnCont := FALSE,
		stConnect := stConnectParam,
		abyData := pSend,
		uiDataSize := UINT#0,
		uiTimeOut := UINT#100,
		xDone => ,
		xBusy => ,
		xError => ,
		wErrorID => ,
		eStatus => ,
		stConnectInfo => );
END_IF;
xSendPrev := i_xSendTrig;

          
END_FUNCTION_BLOCK

PROGRAM PRG_TcpHmi
  VAR
    fbTcp : FB_TCPServer;
    tonWatch : TON;
    tonSend : TON;
    abySend : ARRAY[0..1023] OF BYTE;
    abyRecv : ARRAY[0..1023] OF BYTE;
    strLine : STRING(512);
    strOut : STRING(512);
    i : INT;
    n : INT;
    xSendTrig : BOOL;
    uiSendLen : UINT;
    p : INT;
    xInit : BOOL;
  END_VAR

            (*==============================================================================
 * PRG_TcpHmi — TCP JSON HMI 桥（Server :Tcp_uiPort）
 * 写影子 Tcp_*；读 HMI_Status / AxisFb 组 t:s
 *============================================================================*)
IF NOT xInit THEN
	Tcp_xEStop := TRUE;
	Tcp_rJogVelX := 0.4; Tcp_rSpinVel := 0.3;
	Tcp_rJogVelY := 0.3; Tcp_rJogVelZ := 0.2; Tcp_rJogVelR := 0.2;
	Tcp_rAutoDistX := 1.0; Tcp_rAutoVelX := 0.4;
	Tcp_rAutoVelY := 0.3; Tcp_rAutoVelZ := 0.15;
	Tcp_rWheelBase := 5.0; Tcp_rForceSet := 100.0;
	Tcp_xForceSimEnable := TRUE;
	IF Tcp_uiPort = 0 THEN Tcp_uiPort := 9100; END_IF;
	xInit := TRUE;
END_IF;

fbTcp(
	i_xEnable := TRUE,
	i_uiPort := Tcp_uiPort,
	i_xSendTrig := xSendTrig,
	i_strSend := strOut,
	o_xConnected => Tcp_xConnected,
	o_xRecvNew => ,
	o_strRecv => strLine,
	o_uiRecvLen => ,
	o_xSendDone => ,
	o_xError => ,
	o_wErrorID => );

xSendTrig := FALSE;

IF fbTcp.o_xRecvNew THEN
	(* 心跳 *)
	IF FIND(strLine, '"t":"ping"') > 0 OR FIND(strLine, '"t": "ping"') > 0 THEN
		(* pong 随下次状态发 *)
	END_IF;
	(* BOOL *)
	IF FIND(strLine, '"HMI_xEStop":false') > 0 OR FIND(strLine, '"HMI_xEStop": false') > 0 THEN Tcp_xEStop := FALSE;
	ELSIF FIND(strLine, '"HMI_xEStop":true') > 0 OR FIND(strLine, '"HMI_xEStop": true') > 0 THEN Tcp_xEStop := TRUE; END_IF;
	IF FIND(strLine, '"HMI_xStop":true') > 0 THEN Tcp_xStop := TRUE;
	ELSIF FIND(strLine, '"HMI_xStop":false') > 0 THEN Tcp_xStop := FALSE; END_IF;
	IF FIND(strLine, '"HMI_xStopHold3s":true') > 0 THEN Tcp_xStopHold3s := TRUE;
	ELSIF FIND(strLine, '"HMI_xStopHold3s":false') > 0 THEN Tcp_xStopHold3s := FALSE; END_IF;
	IF FIND(strLine, '"HMI_xStart":true') > 0 THEN Tcp_xStart := TRUE; Tcp_xEnable := TRUE;
	ELSIF FIND(strLine, '"HMI_xStart":false') > 0 THEN Tcp_xStart := FALSE; Tcp_xEnable := FALSE; END_IF;
	IF FIND(strLine, '"HMI_xEnable":true') > 0 THEN Tcp_xEnable := TRUE;
	ELSIF FIND(strLine, '"HMI_xEnable":false') > 0 THEN Tcp_xEnable := FALSE; END_IF;
	IF FIND(strLine, '"HMI_xAutoMode":true') > 0 THEN Tcp_xAutoMode := TRUE;
	ELSIF FIND(strLine, '"HMI_xAutoMode":false') > 0 THEN Tcp_xAutoMode := FALSE; END_IF;
	IF FIND(strLine, '"HMI_xJogXPos":true') > 0 THEN Tcp_xJogXPos := TRUE;
	ELSIF FIND(strLine, '"HMI_xJogXPos":false') > 0 THEN Tcp_xJogXPos := FALSE; END_IF;
	IF FIND(strLine, '"HMI_xJogXNeg":true') > 0 THEN Tcp_xJogXNeg := TRUE;
	ELSIF FIND(strLine, '"HMI_xJogXNeg":false') > 0 THEN Tcp_xJogXNeg := FALSE; END_IF;
	IF FIND(strLine, '"HMI_xSpinLeft":true') > 0 THEN Tcp_xSpinLeft := TRUE;
	ELSIF FIND(strLine, '"HMI_xSpinLeft":false') > 0 THEN Tcp_xSpinLeft := FALSE; END_IF;
	IF FIND(strLine, '"HMI_xSpinRight":true') > 0 THEN Tcp_xSpinRight := TRUE;
	ELSIF FIND(strLine, '"HMI_xSpinRight":false') > 0 THEN Tcp_xSpinRight := FALSE; END_IF;
	IF FIND(strLine, '"HMI_xJogYPos":true') > 0 THEN Tcp_xJogYPos := TRUE;
	ELSIF FIND(strLine, '"HMI_xJogYPos":false') > 0 THEN Tcp_xJogYPos := FALSE; END_IF;
	IF FIND(strLine, '"HMI_xJogYNeg":true') > 0 THEN Tcp_xJogYNeg := TRUE;
	ELSIF FIND(strLine, '"HMI_xJogYNeg":false') > 0 THEN Tcp_xJogYNeg := FALSE; END_IF;
	IF FIND(strLine, '"HMI_xJogZPos":true') > 0 THEN Tcp_xJogZPos := TRUE;
	ELSIF FIND(strLine, '"HMI_xJogZPos":false') > 0 THEN Tcp_xJogZPos := FALSE; END_IF;
	IF FIND(strLine, '"HMI_xJogZNeg":true') > 0 THEN Tcp_xJogZNeg := TRUE;
	ELSIF FIND(strLine, '"HMI_xJogZNeg":false') > 0 THEN Tcp_xJogZNeg := FALSE; END_IF;
	IF FIND(strLine, '"HMI_xJogRPos":true') > 0 THEN Tcp_xJogRPos := TRUE;
	ELSIF FIND(strLine, '"HMI_xJogRPos":false') > 0 THEN Tcp_xJogRPos := FALSE; END_IF;
	IF FIND(strLine, '"HMI_xJogRNeg":true') > 0 THEN Tcp_xJogRNeg := TRUE;
	ELSIF FIND(strLine, '"HMI_xJogRNeg":false') > 0 THEN Tcp_xJogRNeg := FALSE; END_IF;
	IF FIND(strLine, '"HMI_xAutoStart":true') > 0 THEN Tcp_xAutoStart := TRUE;
	ELSIF FIND(strLine, '"HMI_xAutoStart":false') > 0 THEN Tcp_xAutoStart := FALSE; END_IF;
	IF FIND(strLine, '"HMI_xAutoAbort":true') > 0 THEN Tcp_xAutoAbort := TRUE;
	ELSIF FIND(strLine, '"HMI_xAutoAbort":false') > 0 THEN Tcp_xAutoAbort := FALSE; END_IF;
	IF FIND(strLine, '"HMI_xForceSimEnable":true') > 0 THEN Tcp_xForceSimEnable := TRUE;
	ELSIF FIND(strLine, '"HMI_xForceSimEnable":false') > 0 THEN Tcp_xForceSimEnable := FALSE; END_IF;
	(* REAL：网关保证无空格；键后直接数字 *)
	p := FIND(strLine, '"HMI_rJogVelX":');
	IF p > 0 THEN Tcp_rJogVelX := STRING_TO_REAL(MID(strLine, p + 15, 16)); END_IF;
	p := FIND(strLine, '"HMI_rSpinVel":');
	IF p > 0 THEN Tcp_rSpinVel := STRING_TO_REAL(MID(strLine, p + 14, 16)); END_IF;
	p := FIND(strLine, '"HMI_rJogVelY":');
	IF p > 0 THEN Tcp_rJogVelY := STRING_TO_REAL(MID(strLine, p + 15, 16)); END_IF;
	p := FIND(strLine, '"HMI_rJogVelZ":');
	IF p > 0 THEN Tcp_rJogVelZ := STRING_TO_REAL(MID(strLine, p + 15, 16)); END_IF;
	p := FIND(strLine, '"HMI_rJogVelR":');
	IF p > 0 THEN Tcp_rJogVelR := STRING_TO_REAL(MID(strLine, p + 15, 16)); END_IF;
	p := FIND(strLine, '"HMI_rAutoDistX":');
	IF p > 0 THEN Tcp_rAutoDistX := STRING_TO_REAL(MID(strLine, p + 16, 16)); END_IF;
	p := FIND(strLine, '"HMI_rAutoVelX":');
	IF p > 0 THEN Tcp_rAutoVelX := STRING_TO_REAL(MID(strLine, p + 15, 16)); END_IF;
	p := FIND(strLine, '"HMI_rAutoVelY":');
	IF p > 0 THEN Tcp_rAutoVelY := STRING_TO_REAL(MID(strLine, p + 15, 16)); END_IF;
	p := FIND(strLine, '"HMI_rAutoVelZ":');
	IF p > 0 THEN Tcp_rAutoVelZ := STRING_TO_REAL(MID(strLine, p + 15, 16)); END_IF;
	p := FIND(strLine, '"HMI_rWheelBase":');
	IF p > 0 THEN Tcp_rWheelBase := STRING_TO_REAL(MID(strLine, p + 16, 16)); END_IF;
	p := FIND(strLine, '"HMI_rForceSet":');
	IF p > 0 THEN Tcp_rForceSet := STRING_TO_REAL(MID(strLine, p + 15, 16)); END_IF;
	p := FIND(strLine, '"HMI_rForceSim":');
	IF p > 0 THEN Tcp_rForceSim := STRING_TO_REAL(MID(strLine, p + 15, 16)); END_IF;
END_IF;

(* 有接收则本周期 IN=FALSE 复位；否则连接中计时 *)
tonWatch(IN := Tcp_xConnected AND NOT fbTcp.o_xRecvNew, PT := T#500MS);
Tcp_xTimeout := Tcp_xConnected AND tonWatch.Q;
IF Tcp_xTimeout OR NOT Tcp_xConnected THEN
	Tcp_xStop := FALSE; Tcp_xStopHold3s := FALSE;
	Tcp_xStart := FALSE; Tcp_xEnable := FALSE;
	Tcp_xJogXPos := FALSE; Tcp_xJogXNeg := FALSE;
	Tcp_xSpinLeft := FALSE; Tcp_xSpinRight := FALSE;
	Tcp_xJogYPos := FALSE; Tcp_xJogYNeg := FALSE;
	Tcp_xJogZPos := FALSE; Tcp_xJogZNeg := FALSE;
	Tcp_xJogRPos := FALSE; Tcp_xJogRNeg := FALSE;
	Tcp_xAutoStart := FALSE; Tcp_xAutoAbort := FALSE;
	IF Tcp_xTimeout OR NOT Tcp_xConnected THEN Tcp_xEStop := TRUE; END_IF;
END_IF;

tonSend(IN := NOT tonSend.Q, PT := T#100MS);
IF tonSend.Q AND Tcp_xConnected THEN
	strOut := '{"t":"s"';
	strOut := CONCAT(strOut, ',"HMI_eDevState":');
	strOut := CONCAT(strOut, INT_TO_STRING(HMI_eDevState));
	strOut := CONCAT(strOut, ',"HMI_eOpMode":');
	strOut := CONCAT(strOut, INT_TO_STRING(HMI_eOpMode));
	strOut := CONCAT(strOut, ',"HMI_iAutoStepShow":');
	strOut := CONCAT(strOut, INT_TO_STRING(HMI_iAutoStepShow));
	strOut := CONCAT(strOut, ',"HMI_iAlarmShow":');
	strOut := CONCAT(strOut, INT_TO_STRING(HMI_iAlarmShow));
	strOut := CONCAT(strOut, ',"HMI_xDevStop":');
	strOut := CONCAT(strOut, SEL(HMI_xDevStop, 'false', 'true'));
	strOut := CONCAT(strOut, ',"HMI_xDevRun":');
	strOut := CONCAT(strOut, SEL(HMI_xDevRun, 'false', 'true'));
	strOut := CONCAT(strOut, ',"HMI_xDevError":');
	strOut := CONCAT(strOut, SEL(HMI_xDevError, 'false', 'true'));
	strOut := CONCAT(strOut, ',"HMI_xAutoBusy":');
	strOut := CONCAT(strOut, SEL(HMI_xAutoBusy, 'false', 'true'));
	strOut := CONCAT(strOut, ',"HMI_xAutoDone":');
	strOut := CONCAT(strOut, SEL(HMI_xAutoDone, 'false', 'true'));
	strOut := CONCAT(strOut, ',"HMI_xLampEStop":');
	strOut := CONCAT(strOut, SEL(HMI_xLampEStop, 'false', 'true'));
	strOut := CONCAT(strOut, ',"HMI_xLampEnableOk":');
	strOut := CONCAT(strOut, SEL(HMI_xLampEnableOk, 'false', 'true'));
	strOut := CONCAT(strOut, ',"HMI_xLampFault":');
	strOut := CONCAT(strOut, SEL(HMI_xLampFault, 'false', 'true'));
	strOut := CONCAT(strOut, ',"HMI_rForceShow":');
	strOut := CONCAT(strOut, REAL_TO_STRING(HMI_rForceShow));
	strOut := CONCAT(strOut, ',"Tcp_xConnected":true,"Tcp_xTimeout":');
	strOut := CONCAT(strOut, SEL(Tcp_xTimeout, 'false', 'true'));
	strOut := CONCAT(strOut, ',"AxisFb_rPosY":');
	strOut := CONCAT(strOut, REAL_TO_STRING(AxisFb_rPosY));
	strOut := CONCAT(strOut, ',"AxisFb_rPosZ":');
	strOut := CONCAT(strOut, REAL_TO_STRING(AxisFb_rPosZ));
	strOut := CONCAT(strOut, ',"AxisFb_xReady":');
	strOut := CONCAT(strOut, SEL(AxisFb_xReady, 'false', 'true'));
	strOut := CONCAT(strOut, '}');
	strOut := CONCAT(strOut, '$N');
	xSendTrig := TRUE;
END_IF;

          
END_PROGRAM
